TYPE ST_System_BSp_Verb_Zustand :
STRUCT
	Betrieb_Anford		: BOOL;
	Betrieb_Soll			: BOOL;
	Betrieb				: BOOL;

	Freigabe				: BOOL;
	Freigabe_Deakt		: BOOL;
	Freigabe_Code		: WORD;

	Stoerung				: BOOL;
	Stoerung_Code		: WORD;

	Warnung				: BOOL;
	Warnung_Code		: WORD;

	Status					: SINT;
	Status_Vorl_Pumpe		: BOOL;
	Status_Nachl_Pumpe		: BOOL;
	Status_Wiedereinschalten	: BOOL;
	Stoerung_beendet		: BOOL;

	Quittierung			: BOOL;
	Temperaturunterschied	: BOOL;

	Temp_SpeicherA      : REAL;
	Temp_SpeicherB      : REAL;
	Temp_SpeicherC      : REAL;

	Temp_Netz           : REAL;

END_STRUCT
END_TYPE

(* stored: Version 1.1.0.1, ProductVersion 3.1.4024.9
   DUT ST_System_BSp_Verb_Zustand: Id {cc1f6ed7-c492-480c-85a4-13d2bc4404fb} *)
